// Prerun Pump
      A     DB145.DBX  172.6;
      AN    #S2I.SFM37.I00;
      A     #RRel;
      CLR   ;
      =     DB145.DBX  173.3;

// Return Pump
      AN    #Empty;
      A     #RRel;
      =     DB145.DBX  173.4;
      =     DB145.DBX   29.3;

// ---------------------------------------------------------------------------
// control modules (Own CM's)
      A     #ComCIP1;
      A     M    102.3;
      =     DB240.DBX  428.0;

      A     #ComCIP2;
      A     M    102.3;
      =     DB240.DBX  508.0;

      A     #ComCIP3;
      A     M    102.3;
      =     DB240.DBX  588.0;

// Trap Filter
      A     #S2I.SFM14.I01; // Yes
      A     M    102.3;
      CLR   ;
      =     DB240.DBX  188.0;
      =     DB240.DBX  348.0;

      A     #S2I.SFM14.I01; // Yes
      A     M    102.3;
      =     DB240.DBX  268.0;

// ---------------------------------------------------------------------------
// transition condition
//      A     #SubStepMaxD
//      =     "SOPD"


// subphase evaluation
      L     MW   110;
      JL    D500;
      JU    COMM; // subphase  0:
// ---------------------------------------------------------------------------
D500: SET   ;
      S     M    110.7; // Error unknown subphase
      JU    COMM;
NETWORK
TITLE =phase 36: CIP Drain
//SFM   Use                                 Datatype        UoM
//----+-------------------------------------------------------------------------
// 00 : Watch Dog Time                      Duration        Min
// 04 : Delay Empty                         Duration        #sec
X36:  SET   ;
// ---------------------------------------------------------------------------
// General CM evaluation
      CALL FC   140 (
           ChkType                  := 3,
           ChkOK                    := #ChkOK);

      AN    #ChkOK;
      S     M    120.3;

// ---------------------------------------------------------------------------
// general functions
      AN    M    121.2;
      A     M    102.3;
      =     #RRel;

// ---------------------------------------------------------------------------
// messages
// ---------------------------------------------------------------------------
// timer & counter
      A     DB145.DBX  458.5;
      A     M    102.0;
      =     M    130.3;


// ---------------------------------------------------------------------------
// pause timer
      ON    M    102.3;
      O     M    150.3;
      S     M    140.3; // Delay Empty

// ---------------------------------------------------------------------------
// communication

// ---------------------------------------------------------------------------
// control modules
      A     M    102.3;

// ---------------------------------------------------------------------------
// transition condition
      A     M    150.3;
      =     M    102.1;

// subphase evaluation
      L     MW   110;
      JL    D600;
      JU    COMM; // subphase  0:
// ---------------------------------------------------------------------------
D600: SET   ;
      S     M    110.7; // Error unknown subphase
      JU    COMM;
NETWORK
TITLE =phase 38: CIP Randvollstellung
//SFM   Use                                 Datatype        UoM
//----+-------------------------------------------------------------------------
// 00 : Watch Dog Time                      Duration        min
// 01 : Step Time                           Duration        min
// 04 : Delay Level                         Duration        s
// 15 : Amount                              Value           m3
// 17 : Level                               Value           l
// 22 : Agitator Speed                      Value           %
// 27 : CIP Prerun                          Enumeration     min
// 28 : CIP Return                          Enumeration     min
// 29 : CIP Pump Speed                      Value           %
// 34 : CIP Prerun Flow                     Value           m3/h
// 35 : CIP Prerun Pressure                 Value           bar
// 37 : CIP Pump Mode                       Enumeration     min
X38:  SET   ;
// ---------------------------------------------------------------------------
// General CM evaluation
      CALL FC   140 (
           ChkType                  := 3,
           ChkOK                    := #ChkOK);

      AN    #ChkOK;
      S     M    120.3;

// ---------------------------------------------------------------------------
// index evaluation: CIP Prerun
      CALL FC    45 (
           SFM                      := #U.Seq.SFM[27].Sp,
           Indexes                  := #S2I.SFM27);

// ---------------------------------------------------------------------------
// index evaluation: CIP Return
      CALL FC    45 (
           SFM                      := #U.Seq.SFM[28].Sp,
           Indexes                  := #S2I.SFM28);

// ---------------------------------------------------------------------------
// index evaluation: CIP Pump Mode
      CALL FC    45 (
           SFM                      := #U.Seq.SFM[37].Sp,
           Indexes                  := #S2I.SFM37);

// ---------------------------------------------------------------------------
// general functions
      AN    M    121.2;
      A     M    102.3;
      =     #RRel;

// Get Pushout Amount

      A     M    102.2;
      JCN   N381;
      L     #U.Seq.Prop.Val10;
      L     #U.Seq.SFM[15].Sp;
      +R    ;
      T     #U.Seq.SFM[15].Sp;
N381: NOP   0;

// CIP Unit
      AN    #ComCIP;
      ON    DB145.DBX  123.4;
      ON    DB145.DBX  123.5;
      JCN   x381;
      R     #RRel;
      L     949; // CIP Not Ready!
      T     MD    90;
x381: NOP   0;

// CIP Distribution Unit
      AN    #ComCIPDist;
      ON    DB145.DBX  411.4;
      ON    DB145.DBX  411.5;
      JCN   x382;
      R     #RRel;
      L     949; // CIP Partner Not Ready!
      T     MD    90;
x382: NOP   0;

// Partner Unit
      AN    #ComDST;
      ON    DB145.DBX  459.4;
      ON    DB145.DBX  459.5;
      JCN   x383;
      R     #RRel;
      L     903; // Partner Unit Not Ready!
      T     MD    90;
x383: NOP   0;

// CIP Signals ---
      CALL FC   716 (
           StepOnSFMSP              := #U.Seq.SFM[26].Sp,
           EmptySig                 := DB145.DBX  458.5,
           EmptyLevel               := TRUE,
           CIPPumpRun               := DB145.DBX  124.3,
           CIPReady                 := DB145.DBX  123.5,
           Empty                    := #Empty,
           TransCondOK              := M    102.1,
           RRel                     := #RRel);

      A     DB145.DBX  124.3;
      A     M    102.3;
      =     DB145.DBX   29.2;

// ---------------------------------------------------------------------------
// messages
// ---------------------------------------------------------------------------
// timer & counter
// Done in "CIPUnitC"
      A     M    102.3;
      =     M    130.0;
      =     M    131.6;

      A     DB145.DBX  458.2;
      A     M    102.3;
      =     M    130.3;

// ---------------------------------------------------------------------------
// communication
// Active, Prerun & Return
      A     M    102.0;
      =     DB145.DBX  171.4;
      =     DB145.DBX  172.6;
      R     DB145.DBX  172.7;

// Run Release
      A     #RRel;
      =     DB145.DBX  171.5;

// Prerun Pump
      A     DB145.DBX  172.6;
      AN    #S2I.SFM37.I00;
      A     #RRel;
      =     DB145.DBX  173.3;

// Return Pump
      AN    #Empty;
      A     #RRel;
      CLR   ;
      =     DB145.DBX  173.4;
      =     DB145.DBX   29.3;

// ---------------------------------------------------------------------------
// control modules (Own CM's)
      A     #ComCIP1;
      A     M    102.3;
      =     DB240.DBX  428.0;

      A     #ComCIP2;
      A     M    102.3;
      =     DB240.DBX  508.0;

      A     #ComCIP3;
      A     M    102.3;
      =     DB240.DBX  588.0;

// Trap Filter
      A     #S2I.SFM14.I01; // Yes
      A     M    102.3;
      CLR   ;
      =     DB240.DBX  188.0;
      =     DB240.DBX  348.0;

      A     #S2I.SFM14.I01; // Yes
      A     M    102.3;
      =     DB240.DBX  268.0;

// ---------------------------------------------------------------------------
// transition condition
      A     M    150.3;
      =     M    102.1;


// Nach Randvollstellung nach "CIP Ende"
      L     #U.Seq.StepMax; // CIP Ende = letzter Schritt
      T     MW   106;

// subphase evaluation
      L     MW   110;
      JL    D800;
      JU    COMM; // subphase  0:
// ---------------------------------------------------------------------------
D800: SET   ;
      S     M    110.7; // Error unknown subphase
      JU    COMM;
NETWORK
TITLE =phase 39: CIP Rinsing from RWT
//SFM   Use                                 Datatype        UoM
//----+-------------------------------------------------------------------------
// 00 : Watch Dog Time                      Duration        min
// 01 : Step Time                           Duration        min
// 05 : Substep Time                        Duration        s
// 06 : Delay Switchpoint                   Duration        s
// 15 : Amount                              Value           m3
// 27 : CIP Prerun                          Enumeration     min
// 28 : CIP Return                          Enumeration     min
// 29 : CIP Pump Speed                      Value           %
// 30 : CIP Return Temperature              Value           °C
// 32 : CIP Return Conductivity             Value           mS
// 34 : CIP Prerun Flow                     Value           m3/h
// 35 : CIP Prerun Pressure                 Value           bar
// 37 : CIP Pump Mode                       Enumeration     min
// 59 : Interval Counter                    Value           No.
X39:  SET   ;
// ---------------------------------------------------------------------------
// General CM evaluation
      CALL FC   140 (
           ChkType                  := 3,
           ChkOK                    := #ChkOK);

      AN    #ChkOK;
      S     M    120.3;

// ---------------------------------------------------------------------------
// index evaluation: CIP Prerun
      CALL FC    45 (
           SFM                      := #U.Seq.SFM[27].Sp,
           Indexes                  := #S2I.SFM27);

// ---------------------------------------------------------------------------
// index evaluation: CIP Return
      CALL FC    45 (
           SFM                      := #U.Seq.SFM[28].Sp,
           Indexes                  := #S2I.SFM28);

// ---------------------------------------------------------------------------
// index evaluation: CIP Pump Mode
      CALL FC    45 (
           SFM                      := #U.Seq.SFM[37].Sp,
           Indexes                  := #S2I.SFM37);

// ---------------------------------------------------------------------------
// general functions
      AN    M    121.2;
      A     M    102.3;
      =     #RRel;

// CIP Unit
      AN    #ComCIP;
      ON    DB145.DBX  123.4;
      ON    DB145.DBX  123.5;
      JCN   x391;
      R     #RRel;
      L     949; // CIP Not Ready!
      T     MD    90;
x391: NOP   0;

// CIP Distribution Unit
      AN    #ComCIPDist;
      ON    DB145.DBX  411.4;
      ON    DB145.DBX  411.5;
      JCN   x392;
      R     #RRel;
      L     949; // CIP Partner Not Ready!
      T     MD    90;
x392: NOP   0;

// Partner Unit
      AN    #ComDST;
      ON    DB145.DBX  459.4;
      ON    DB145.DBX  459.5;
      JCN   x393;
      R     #RRel;
      L     903; // Partner Unit Not Ready!
      T     MD    90;
x393: NOP   0;

// CIP Signals ---
      CALL FC   716 (
           StepOnSFMSP              := #U.Seq.SFM[26].Sp,
           EmptySig                 := DB145.DBX  458.5,
           EmptyLevel               := TRUE,
           CIPPumpRun               := DB145.DBX  124.3,
           CIPReady                 := DB145.DBX  123.5,
           Empty                    := #Empty,
           TransCondOK              := M    102.1,
           RRel                     := #RRel);


      A     DB145.DBX  124.3;
      A     M    102.3;
      =     DB145.DBX   29.2;



// ---------------------------------------------------------------------------
// messages
// ---------------------------------------------------------------------------
// timer & counter
// Done in "CIPUnitC"

// ---------------------------------------------------------------------------
// pause timer
      ON    M    102.3;
      O     M    150.0;
      S     M    140.0; // Step Time

      ON    M    102.3;
      O     M    150.5;
      S     M    140.5; // Delay Switchpoint

// ---------------------------------------------------------------------------
// communication
// Active, Prerun & Return
      A     M    102.0;
      =     DB145.DBX  171.4;
      =     DB145.DBX  172.7;
      =     DB145.DBX  172.6;

// Run Release
      A     #RRel;
      =     DB145.DBX  171.5;

// Prerun Pump
      A     DB145.DBX  459.5;
      A     DB145.DBX  172.6;
      AN    #S2I.SFM37.I00;
      A     #RRel;
      =     DB145.DBX  173.3;

// Return Pump
      AN    #Empty;
      A     #RRel;
      =     DB145.DBX  173.4;
      =     DB145.DBX   29.3;

// Mit Abluaf
      AN    M    157.2;
      A     M    102.0;
      =     DB145.DBX   29.5;

// ---------------------------------------------------------------------------
// control modules (Own CM's)
      A     #ComCIP1;
      A     M    102.3;
      =     DB240.DBX  428.0;

      A     #ComCIP2;
      A     M    102.3;
      =     DB240.DBX  508.0;

      A     #ComCIP3;
      A     M    102.3;
      =     DB240.DBX  588.0;

// Trap Filter
      A     #S2I.SFM14.I01; // Yes
      A     M    102.3;
      CLR   ;
      =     DB240.DBX  188.0;
      =     DB240.DBX  348.0;

      A     #S2I.SFM14.I01; // Yes
      A     M    102.3;
      =     DB240.DBX  268.0;

// ---------------------------------------------------------------------------
// transition condition
//      A     #SubStepMaxD
//      =     "SOPD"

// ---------------------------------------------------------------------------
// ---------------------------------------------------------------------------
// subphase repeat function
      A     #SubStepMax;
      JCN   Y39;
      L     1;
      T     MW   116;
Y39:  SET   ;

      A     #SubStepMax;
      AN    M    103.0;
      JCN   Y39a;
      L     #U.Seq.SFM[59].Val; // Increment Interval Counter
      L     1.000000e+000;
      +R    ;
      T     #U.Seq.SFM[59].Val;
Y39a: SET   ;
      A     M    102.2;
      ON    M    102.0;
      JCN   In2R; // Reset Interval Counter at Start and End Of Phase
      L     0.000000e+000;
      T     #U.Seq.SFM[59].Val;
In2R: NOP   0;

// subphase evaluation
      L     MW   110;
      JL    D900;
      JU    COMM; // subphase  0:
      JU    D901; // subphase  1: Pause
      JU    D902; // subphase  2: Main
      JU    D903; // subphase  3: Expulse
      JU    D904; // subphase  4: Seat Lift
      JU    D900; // subphase  5:
      JU    D906; // subphase  6: Shaft Rinse
      JU    D907; // subphase  7: Drain
// ---------------------------------------------------------------------------
D900: SET   ;
      S     M    110.7; // Error unknown subphase
      JU    COMM;

// subphase 1: Pause
D901: SET   ;

      A     M    103.0;
      R     DB145.DBX  173.3;

// -------------------------------------------------
// subphase timer & counter
      A     M    103.0;
      =     M    130.4; // Substep Time
// -------------------------------------------------
// subphase actuator

// -------------------------------------------------
// subphase transition
      A     M    150.3; // Delay Level
      A     M    130.3;
      O     M    150.4; // Substep Time Done
      =     M    103.1;
      JU    COMM;

// subphase 2: Main
D902: SET   ;

// -------------------------------------------------
// subphase timer & counter
      A     M    103.0;
      =     M    130.4; // Substep Time

// -------------------------------------------------
// subphase actuator
      A     M    103.3;


// -------------------------------------------------
// subphase transition
      A     M    150.4; // Substep Time Done
      =     M    103.1;
      JU    COMM;

// subphase 3: Expulse
D903: SET   ;

// -------------------------------------------------
// subphase timer & counter
      A     M    103.0;

// -------------------------------------------------
// subphase actuator
      A     M    103.3;

// -------------------------------------------------
// subphase transition
      CLR   ;
      =     M    103.1;
      JU    COMM;

// subphase 4: Seat Lift
D904: SET   ;

// -------------------------------------------------
// subphase timer & counter
      A     M    103.0;

// -------------------------------------------------
// subphase actuator
      A     M    103.3;

// -------------------------------------------------
// subphase transition
      SET   ;
      =     M    103.1;
      JU    COMM;

// subphase 6: Shaft Rinse
D906: SET   ;

// -------------------------------------------------
// subphase timer & counter
      A     M    103.0;
      =     M    130.4; // Substep Time

// -------------------------------------------------
// subphase actuator
      A     M    103.3;
      =     DB240.DBX  668.0;

// -------------------------------------------------
// subphase transition
      A     M    150.4; // Substep Time Done
      O     M    157.2; // Interval Counter Done
      =     M    103.1;
      JU    COMM;

// subphase 7: Drain
D907: SET   ;

// -------------------------------------------------
// subphase timer & counter
      A     M    103.0;
      =     M    130.4; // Substep Time

// -------------------------------------------------
// subphase actuator
      A     M    103.3;
      R     DB145.DBX  173.6; // Req Drain RV1_RS
      R     DB145.DBX   29.6; // Req Common Drain
      R     DB2990.DBX  268.0;

// -------------------------------------------------
// subphase transition
      A     M    150.4; // Substep Time Done
      O     M    157.2; // Interval Counter Done
      =     M    103.1;
      JU    COMM;
NETWORK
TITLE =phase 40: CIP End
//SFM   Use                                 Datatype        UoM
//----+-------------------------------------------------------------------------
// 00 : Watch Dog Time                      Duration        min
X40:  SET   ;
// ---------------------------------------------------------------------------
// General CM evaluation
      CALL FC   140 (
           ChkType                  := 3,
           ChkOK                    := #ChkOK);

      AN    #ChkOK;
      S     M    120.3;

// ---------------------------------------------------------------------------
// general functions
//      AN    "SOSTAl"
      A     M    102.3;
      =     #RRel;

// CIP Signals ---
      CALL FC   716 (
           StepOnSFMSP              := 0.000000e+000,
           EmptySig                 := FALSE,
           EmptyLevel               := FALSE,
           CIPPumpRun               := FALSE,
           CIPReady                 := FALSE,
           Empty                    := #xTmp,
           TransCondOK              := #xTmp,
           RRel                     := #RRel);

// ---------------------------------------------------------------------------
// communication
      A     M    102.0;
      =     DB145.DBX   29.7;
      =     DB145.DBX  173.7;

// ---------------------------------------------------------------------------
// transition condition
      AN    #ComCIP;
      AN    #ComCIPDist;
      AN    #ComDST;
      =     M    102.1;


// subphase evaluation
      L     MW   110;
      JL    E000;
      JU    COMM; // subphase  0:
// ---------------------------------------------------------------------------
E000: SET   ;
      S     M    110.7; // Error unknown subphase
      JU    COMM;

NETWORK
TITLE =End Of Sequence Organisation

COMM: SET   ;

// ---------------------------------------------------------------------------
// pause timer unit parameter


NETWORK
TITLE =General Post Phase Controls

      NOP   0;

// ---------------------------------------------------------------------------
// general postphase controls

      L     #U.Seq.PrId;
      L     DB1945.DBD   10;
      ==D   ;
      A(    ;
      L     0;
      >D    ;
      )     ;
      JCN   CIP1;

      CALL SFC   20 (
           SRCBLK                   := DB145.ToCIP,
           RET_VAL                  := #iTmp,
           DSTBLK                   := DB502.ToCIP1);

CIP1: NOP   0;

      L     #U.Seq.PrId;
      L     DB1955.DBD   10;
      ==D   ;
      A(    ;
      L     0;
      >D    ;
      )     ;
      JCN   CIP2;

      CALL SFC   20 (
           SRCBLK                   := DB145.ToCIP,
           RET_VAL                  := #iTmp,
           DSTBLK                   := DB502.ToCIP2);
CIP2: NOP   0;

      L     #U.Seq.PrId;
      L     DB1965.DBD   10;
      ==D   ;
      A(    ;
      L     0;
      >D    ;
      )     ;
      JCN   CIP3;

      CALL SFC   20 (
           SRCBLK                   := DB145.ToCIP,
           RET_VAL                  := #iTmp,
           DSTBLK                   := DB502.ToCIP3);

CIP3: NOP   0;


// Check Selection / Material -----------------------------------------------
      L     0;
      L     DB145.DBD  222; // 1. Tank
      <R    ;
      JCN   MCk1;
      L     #U.Seq.SFM[42].Sp;
      <>R   ;
      S     M    120.3;
      JCN   MCk0;
      L     910;
      T     MD    80;
MCk0: NOP   0;
      L     0;
      L     DB145.DBD  270; // 1. Tank
      <R    ;
      JCN   MCk1;
      L     #U.Seq.SFM[42].Sp;
      <>R   ;
      JCN   MCk1;
      L     910;
      T     MD    90;
MCk1: NOP   0;
      L     0;
      L     DB145.DBD  318; // 2. Tank
      <R    ;
      JCN   MCk2;
      L     #U.Seq.SFM[42].Sp;
      <>R   ;
      JCN   MCk2;
      L     910;
      T     MD    90;
MCk2: NOP   0;
      L     0;
      L     DB145.DBD  366; // 3. Tank
      <R    ;
      JCN   MCk3;
      L     #U.Seq.SFM[42].Sp;
      <>R   ;
      JCN   MCk3;
      L     910;
      T     MD    90;
MCk3: NOP   0;

      L     #U.Seq.SFM[11].Sp;
      L     #U.Seq.SFM[12].Sp;
      OD    ;
      L     #U.Seq.SFM[13].Sp;
      OD    ;
      L     0;
      >R    ;
      O     M    120.7;
      O     #CIP;
      JC    TSel;
      L     906; // "Source not Selected"
      T     MD    90;
TSel: NOP   0;

NETWORK
TITLE =Process Status Management

      NOP   0;
// ---------------------------------------------------------------------------
// Signal Control

      OPN   DB   500;
      L     #UnitNo;
      L     32; //U Structure Length
      *I    ;
      L     20; //DB Heading Offset
      +I    ;
      SLD   3;
      LAR2  ;

// -------------------------------------------------
// Maintenance
      A     #U.Seq.Switch.Sw31;
      OPN   DB   500;
      =     DBX [AR2,P#0.0]; //"PStatD".U[#UnitNo].MTNC
// -------------------------------------------------
// CIP Required
// -------------------------------------------------
// CIP Active
// -------------------------------------------------
// CIP Clean
// -------------------------------------------------
// SIP Required
// -------------------------------------------------
// SIP Active
// -------------------------------------------------
// SIP Clean
// -------------------------------------------------
// Full
      A     DB145.DBX   26.2;
      OPN   DB   500;
      =     DBX [AR2,P#0.7]; //"PStatD".U[#UnitNo].FULL
// -------------------------------------------------
// Filling
      A     DB145.DBX   26.1;
      OPN   DB   500;
      =     DBX [AR2,P#1.0]; //"PStatD".U[#UnitNo].FILL
// -------------------------------------------------
// Ready For Filling
      A     DB145.DBX   26.0;
      OPN   DB   500;
      =     DBX [AR2,P#1.1]; //"PStatD".U[#UnitNo].RFFI
// -------------------------------------------------
// Empty
      A     DB145.DBX   26.5;
      OPN   DB   500;
      =     DBX [AR2,P#1.2]; //"PStatD".U[#UnitNo].EMTY
// -------------------------------------------------
// Emptying
      A     DB145.DBX   26.4;
      OPN   DB   500;
      =     DBX [AR2,P#1.3]; //"PStatD".U[#UnitNo].EMTI
// -------------------------------------------------
// Ready For Emptying
      A     DB145.DBX   26.3;
      OPN   DB   500;
      =     DBX [AR2,P#1.4]; //"PStatD".U[#UnitNo].RFEM
// -------------------------------------------------
// Reserved
//      A     #ComXYZ
//      OPN   "PStatD"
//      =     DBX [AR2,P#1.5]             //"PStatD".U[#UnitNo].RESV
// -------------------------------------------------
// Production
// -------------------------------------------------
// Used

// -------------------------------------------------
// PStat Function Call

      CALL FC   500 (
           UnitNo                   := #UnitNo,
           PStatModVal              := DB245.DBD  234);



NETWORK
TITLE =Unit Hold Request and Messages

      SET   ;

// ---------------------------------------------------------------------------
// Set unit to "hold" if maintenance
      AN    #U.Seq.Switch.Sw31; // maintenance !
      JC    NCO1;
      S     M    120.3;
      L     998; // "Unit in maintenance !"
      T     MD    90;

// ---------------------------------------------------------------------------
// Set unit to "hold" if emergency stop
NCO1: A     #EStopOK;
      JC    NCO2;
      S     M    120.3;
      L     999; // "Emergency stop !"
      T     MD    90;
NCO2: NOP   0;

// ---------------------------------------------------------------------------
// Check Partner
      AN    #S2I.SFM10.I00;
      AN    #U.Seq.PO.B22;
      AN    #U.Seq.Step0;
      AN    #CIP;
      =     #xTmp;


      AN    DB145.DBX  218.3;
      AN    DB145.DBX  218.4;
      A     #xTmp;
      JCN   NC03;
      L     904; // "Source Not Ready!
      T     MD    90;
NC03: NOP   0;

      AN    DB145.DBX  218.3;
      ON    DB145.DBX  218.4;
      AN    #ComSRC;
      AN    #U.Seq.Step0;
      AN    #U.Seq.PO.B22;
      AN    #CIP;
      JCN   NC06;
      L     909; // Source for Material not found
      T     MD    90;
NC06: NOP   0;

      AN    #S2I.SFM14.I02;
      AN    #U.Seq.Step0;
      AN    #CIP;
      CLR   ;
      JCN   NC04;
      L     903; // Partner not Ready
      T     MD    90;
NC04: NOP   0;

      AN    DB145.DBX  458.0; // Water Tank Ready
      AN    DB145.DBX  458.1;
      AN    #U.Seq.Step0;
      AN    #U.Seq.PO.B3;
      AN    #CIP;
      CLR   ;
      JCN   NC05;
      L     903; // Destination not Ready
      T     MD    90;
NC05: NOP   0;






END_FUNCTION_BLOCK

FUNCTION_BLOCK FB 143
TITLE =C04: Water Transfer Plant x
AUTHOR : Woermann
FAMILY : BOTEC_F1
NAME : C04E
VERSION : 1.2
CODE_VERSION1


VAR
  U : UDT 141;
END_VAR
VAR_TEMP
  CIP : BOOL ;	//CIP active
  UNIM : BOOL ;	//Unit Not In Maintenance
  GenRel : BOOL ;	//general OK (emergency and maintenance OK)
  EStopOK : BOOL ;	//emergency OK
  UnitNo : INT ;	//unit number
  xTmp : BOOL ;	//Temporary Bool
  iTmp : INT ;	//Temporary INT
  rTmp : REAL ;	//Temporary REAL
  dTmp : DINT ;	//Temporary DINT (free for general use)
  RetValInt : INT ;	//return value
  ComCIP1 : BOOL ;	//CIP1 in use
  ComCIP3 : BOOL ;	//CIP3 in use
END_VAR
BEGIN
NETWORK
TITLE =General

      SET   ;
// Simulation ---------------------------------------------------------------
      A     #U.Seq.User.Bit63;
      CC    FB   149; // "C04Sim"
      A     #U.Seq.Sim;
      =     #U.Seq.User.Bit63; //Help bit for simulation

// get unit number ----------------------------------------------------------
      L     #U.Seq.UnitNo;
      T     #UnitNo;

// CIP ----------------------------------------------------------------------
      L     #U.Seq.ProgNo;
      L     0;
      <D    ;
      =     #CIP;

// emergency OK -------------------------------------------------------------
      A     DB145.DBX   27.0; //Emergency Stop OK
      =     #EStopOK;

// Write Unit in Maintenance ------------------------------------------------

      AN    #U.Seq.Switch.Sw31;
      =     #UNIM;

// emergency and maintenance OK ---------------------------------------------
      A     #EStopOK;
      A     #UNIM;
      =     #GenRel;

// communication ------------------------------------------------------------
      UC    FB   145; // C04Com

NETWORK
TITLE =Universal Value

      NOP   0;

// ----------------------------------------------------------
// unv001 Process Status
// ----------------------------------------------------------
// process value to UnV
//      L     0.000000e+000
//      T     "C04UnVD".unv001.ValExt

// ----------------------------------------------------------
// unv002 Universal Value 02
// ----------------------------------------------------------
// process value to UnV
//      L     0.000000e+000
//      T     "C04UnVD".unv002.ValExt

// ----------------------------------------------------------
// unv003 Universal Value 03
// ----------------------------------------------------------
// process value to UnV
//      L     0.000000e+000
//      T     "C04UnVD".unv003.ValExt

// ----------------------------------------------------------
// unv004 Universal Value 04
// ----------------------------------------------------------
// process value to UnV
//      L     0.000000e+000
//      T     "C04UnVD".unv004.ValExt

NETWORK
TITLE =Special Input

      NOP   0;

// ----------------------------------------------------------
// RM_KEG_V14 KEG_V14
// ----------------------------------------------------------
      CLR   ;
      =     DB241.DBX   81.4;
      =     DB241.DBX   81.5;

NETWORK
TITLE =Messages

      NOP   0;

// ----------------------------------------------------------
// msg001 Message 01
// ----------------------------------------------------------
      SET   ;
      R     DB247.DBX   80.7;
      =     DB247.DBX   81.4;

      CLR   ;
      =     DB247.DBX   82.7;

// ----------------------------------------------------------
// msg002 Message 02
// ----------------------------------------------------------
      SET   ;
      R     DB247.DBX  140.7;
      =     DB247.DBX  141.4;

      CLR   ;
      =     DB247.DBX  142.7;

// ----------------------------------------------------------
// msg003 Message 03
// ----------------------------------------------------------
      SET   ;
      R     DB247.DBX  200.7;
      =     DB247.DBX  201.4;

      CLR   ;
      =     DB247.DBX  202.7;

NETWORK
TITLE =Sequence organisation


// SFM supply ----------------------------------------------------------------


NETWORK
TITLE =Auto / Manual

      SET   ;
      AN    M    122.2;
      JC    MODE;
      AN    M    120.1;

// assign actuator mode
      AN    M    120.1;
      =     DB240.DBX  105.4;
      =     DB240.DBX  185.4;
      =     DB240.DBX  265.4;
      =     DB240.DBX  345.4;
      =     DB240.DBX  425.4;
      =     DB240.DBX  505.4;
      =     DB240.DBX  585.4;
      =     DB240.DBX  665.4;
      =     DB240.DBX  745.4;
      =     DB240.DBX  825.4;
MODE: SET   ;

NETWORK
TITLE =Wasserpumpe
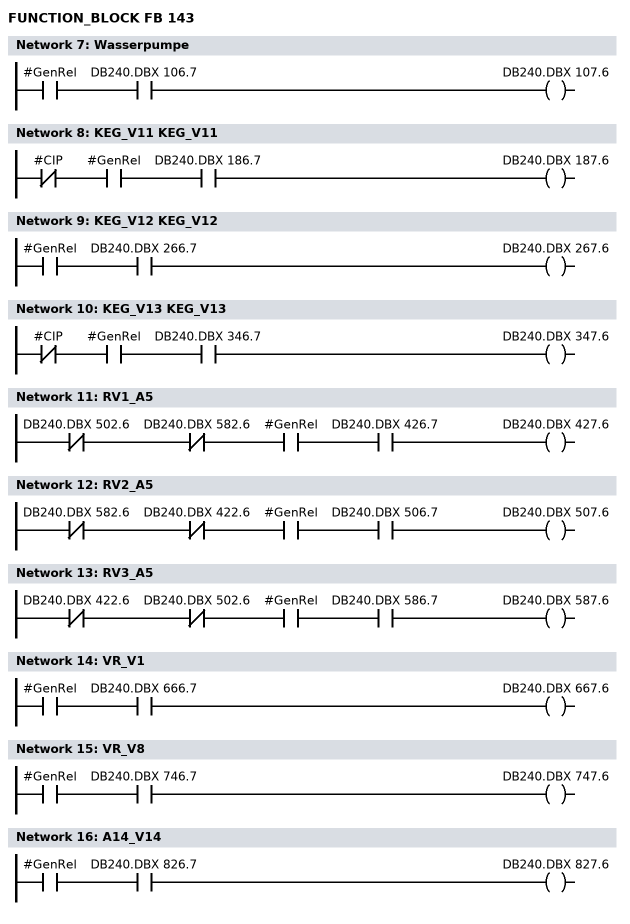

      A     #GenRel;
      A     DB240.DBX  106.7;
      =     DB240.DBX  107.6;

NETWORK
TITLE =KEG_V11 KEG_V11

      AN    #CIP;
      A     #GenRel;
      A     DB240.DBX  186.7;
      =     DB240.DBX  187.6;
NETWORK
TITLE =KEG_V12 KEG_V12

      A     #GenRel;
      A     DB240.DBX  266.7;
      =     DB240.DBX  267.6;
NETWORK
TITLE =KEG_V13 KEG_V13

      AN    #CIP;
      A     #GenRel;
      A     DB240.DBX  346.7;
      =     DB240.DBX  347.6;
NETWORK
TITLE =RV1_A5

      AN    DB240.DBX  502.6;
      AN    DB240.DBX  582.6;

      A     #GenRel;
      A     DB240.DBX  426.7;
      =     DB240.DBX  427.6;

NETWORK
TITLE =RV2_A5

      AN    DB240.DBX  582.6;
      AN    DB240.DBX  422.6;

      A     #GenRel;
      A     DB240.DBX  506.7;
      =     DB240.DBX  507.6;

NETWORK
TITLE =RV3_A5

      AN    DB240.DBX  422.6;
      AN    DB240.DBX  502.6;

      A     #GenRel;
      A     DB240.DBX  586.7;
      =     DB240.DBX  587.6;

NETWORK
TITLE =VR_V1

      A     #GenRel;
      A     DB240.DBX  666.7;
      =     DB240.DBX  667.6;

NETWORK
TITLE =VR_V8

      A     #GenRel;
      A     DB240.DBX  746.7;
      =     DB240.DBX  747.6;

NETWORK
TITLE =A14_V14

      A     #GenRel;
      A     DB240.DBX  826.7;
      =     DB240.DBX  827.6;

END_FUNCTION_BLOCK

FUNCTION_BLOCK FB 145
TITLE =C04: Water Transfer Plant x
AUTHOR : Woermann
FAMILY : BOTEC_F1
NAME : C04Comm
VERSION : 0.1
CODE_VERSION1


VAR
  U : UDT 141;
END_VAR
VAR_TEMP
  iRetVal : INT ;	//return value as integer
  wRetVal : WORD ;	//return value as word
  Run : BOOL ;	//Unit in "RUN" mode
  EStopOK : BOOL ;	//Emergency Stop OK
  CIP : BOOL ;	//CIP Program Selected
  ComCIP : BOOL ;	//Communication with CIP Active
  xTmp : BOOL ;	//Temporary BOOL (free for general use)
  iTmp : INT ;	//Temporary INT (free for general use)
  rTmp : REAL ;	//Temporary REAL (free for general use)
  dTmp : DINT ;	//Temporary DINT (free for general use)
  UnitNo : INT ;	//Unit Number
  EquipmentID : INT ;	//Equipment ID
  Prid : DINT ;	//Process ID
  SFM36 : STRUCT 	//CIP Pump Mode
   I00 : BOOL ;	// Off
   I01 : BOOL ;	// Flow
   I02 : BOOL ;	// Pressure
   I03 : BOOL ;	// Fix Speed
   I04 : BOOL ;
   I05 : BOOL ;
   I06 : BOOL ;
   I07 : BOOL ;
   I08 : BOOL ;
   I09 : BOOL ;
   I10 : BOOL ;
   I11 : BOOL ;
   I12 : BOOL ;
   I13 : BOOL ;
   I14 : BOOL ;
   I15 : BOOL ;
   I16 : BOOL ;
   I17 : BOOL ;
   I18 : BOOL ;
   I19 : BOOL ;
   I20 : BOOL ;
   I21 : BOOL ;
   I22 : BOOL ;
   I23 : BOOL ;
   I24 : BOOL ;
   I25 : BOOL ;
   I26 : BOOL ;
   I27 : BOOL ;
   I28 : BOOL ;
   I29 : BOOL ;
   I30 : BOOL ;
   I31 : BOOL ;
  END_STRUCT ;
  iPLC : INT ;
  iUnit : INT ;
  rUnitNo : REAL ;
  DSTUnit : INT ;	//Destination Unit
  SRCUnit : INT ;
  STBYUnit : INT ;
  rEquipmentID : REAL ;
  dst0 : BOOL ;	//No Destination Selected
END_VAR
BEGIN
NETWORK
TITLE =general

      SET   ;

// unit & equipment number ---------------------------------------------------
      L     #U.Seq.UnitNo;
      T     #UnitNo;

      L     DB145.DBW   14;
      L     1000;
      *I    ;
      L     #UnitNo;
      +I    ;
      T     #EquipmentID;

      L     #EquipmentID;
      ITD   ;
      DTR   ;
      T     #rEquipmentID;

// CIP ----------------------------------------------------------------------
      L     DB145.DBW   18;
      L     0;
      <I    ;
      =     #CIP;

// Communicating Units-------------------------------------------------------
      L     DB145.DBD   10;
      L     DB145.DBD  106;
      ==D   ;
      =     #ComCIP;


NETWORK
TITLE =read other unit's data

      SET   ;

// ... General Unit ----------/

      CALL SFC   20 (
           SRCBLK                   := DB1995.Own,
           RET_VAL                  := #iRetVal,
           DSTBLK                   := DB145.GEN);

// emergency OK -------------------------------------------------------------
      A     DB145.DBX   75.0; //General Emergency Stop OK
      =     #EStopOK;


//----------------------------------------
// Communication Water Tank
//----------------------------------------

// Current Tank ----------------------------

      L     #U.Seq.SFM[10].Sp;
      L     0.000000e+000;
      >R    ;
      JCN   N201;

      CALL FC   950 (
           EquipmentNo              := #U.Seq.SFM[10].Sp,
           PLCNo                    := #iPLC,
           UnitNo                   := #iUnit);

      CALL FC   563 (
           ActReq                   := M    101.0,
           PLCNo                    := #iPLC,
           SourceUnitNo             := #iUnit,
           IsTUnit                  := FALSE,
           DstComDRec               := DB145.SRC,
           RET_VAL                  := #wRetVal);
      JU    N2x1;
N201: NOP   0;
      L     0;
      T     #rTmp;
      CALL SFC   21 (
           BVAL                     := #rTmp,
           RET_VAL                  := #iTmp,
           BLK                      := DB145.SRC);
N2x1: NOP   0;

// Priority 1 -----------------------------

      L     #U.Seq.SFM[11].Sp;
      L     0.000000e+000;
      >R    ;
      JCN   N202;


      CALL FC   950 (
           EquipmentNo              := #U.Seq.SFM[11].Sp,
           PLCNo                    := #iPLC,
           UnitNo                   := #iUnit);

      CALL FC   563 (
           ActReq                   := M    101.0,
           PLCNo                    := #iPLC,
           SourceUnitNo             := #iUnit,
           IsTUnit                  := FALSE,
           DstComDRec               := DB145.SRC1,
           RET_VAL                  := #wRetVal);
      JU    N2x2;
N202: NOP   0;
      L     0;
      T     #rTmp;
      CALL SFC   21 (
           BVAL                     := #rTmp,
           RET_VAL                  := #iTmp,
           BLK                      := DB145.SRC1);
N2x2: NOP   0;

// Priority 2 ----------------------------

      L     #U.Seq.SFM[12].Sp;
      L     0.000000e+000;
      >R    ;
      JCN   N203;


      CALL FC   950 (
           EquipmentNo              := #U.Seq.SFM[12].Sp,
           PLCNo                    := #iPLC,
           UnitNo                   := #iUnit);

      CALL FC   563 (
           ActReq                   := M    101.0,
           PLCNo                    := #iPLC,
           SourceUnitNo             := #iUnit,
           IsTUnit                  := FALSE,
           DstComDRec               := DB145.SRC2,
           RET_VAL                  := #wRetVal);
      JU    N2x3;
N203: NOP   0;
      L     0;
      T     #rTmp;
      CALL SFC   21 (
           BVAL                     := #rTmp,
           RET_VAL                  := #iTmp,
           BLK                      := DB145.SRC2);
N2x3: NOP   0;

// Priority 3 ----------------------------

      L     #U.Seq.SFM[13].Sp;
      L     0.000000e+000;
      >R    ;
      JCN   N204;


      CALL FC   950 (
           EquipmentNo              := #U.Seq.SFM[13].Sp,
           PLCNo                    := #iPLC,
           UnitNo                   := #iUnit);

      CALL FC   563 (
           ActReq                   := M    101.0,
           PLCNo                    := #iPLC,
           SourceUnitNo             := #iUnit,
           IsTUnit                  := FALSE,
           DstComDRec               := DB145.SRC3,
           RET_VAL                  := #wRetVal);
      JU    N2x4;
N204: NOP   0;
      L     0;
      T     #rTmp;
      CALL SFC   21 (
           BVAL                     := #rTmp,
           RET_VAL                  := #iTmp,
           BLK                      := DB145.SRC3);
N2x4: NOP   0;

//----------------------------------------
// Communication Packaging Plant
//----------------------------------------
      L     #U.Seq.Prop.Index0; // Destination
      ITD   ;
      DTR   ;
      T     #rTmp;

      CALL FC   950 (
           EquipmentNo              := #rTmp,
           PLCNo                    := #iPLC,
           UnitNo                   := #iUnit);


      CALL FC   563 (
           ActReq                   := M    101.0,
           PLCNo                    := #iPLC,
           SourceUnitNo             := #iUnit,
           IsTUnit                  := FALSE,
           DstComDRec               := DB145.DST,
           RET_VAL                  := #wRetVal);

NETWORK
TITLE =external releases

      SET   ;
      =     DB240.DBX  106.7;
      =     DB240.DBX  186.7;
      =     DB240.DBX  266.7;
      =     DB240.DBX  346.7;
      =     DB240.DBX  426.7;
      =     DB240.DBX  506.7;
      =     DB240.DBX  586.7;
      =     DB240.DBX  666.7;
      =     DB240.DBX  746.7;
      =     DB240.DBX  826.7;

NETWORK
TITLE =write own unit data

      SET   ;

//-- CIP Communication ---------------------------------------
      AN    #U.Seq.Step0;
      AN    #U.Seq.PO.B30; // CIP Active (Slave)
      O(    ;
      A     #U.Seq.PO.B3; // Prerinse
      L     DB145.DBD   10;
      L     DB145.DBD  394;
      ==I   ;
      )     ;
//    A     #ComCIP
      JCN   NCIP;
//Conductivity CIP Return
      L     DB145.DBD  150;
      T     #U.Seq.SFM[32].Val;

//Temperature CIP Return
      L     DB145.DBD  146;
      T     #U.Seq.SFM[30].Val;

//CIP Prerun Pump SP

      CALL FC    45 (
           SFM                      := #U.Seq.SFM[36].Sp,
           Indexes                  := #SFM36);


      L     0.000000e+000;
      A     #SFM36.I01;
      =     DB145.DBX  171.7;
      JCN   pfc;
      L     #U.Seq.SFM[34].Sp;
pfc:  NOP   0;
      A     #SFM36.I02;
      =     DB145.DBX  172.0;
      JCN   ppc;
      L     #U.Seq.SFM[35].Sp;
ppc:  NOP   0;
      A     #SFM36.I03;
      =     DB145.DBX  171.6;
      JCN   pxc;
      L     #U.Seq.SFM[29].Sp;
pxc:  NOP   0;
      T     DB145.DBD  182;

// CIP Prerun Temperature
      L     #U.Seq.SFM[36].Sp;
      T     DB145.DBD  182;

//CIP Return
      L     #U.Seq.SFM[28].Sp;
      T     DB145.DBD  186;
      L     DB145.DBD  138;
      T     #U.Seq.SFM[28].Val;

//CIP Prerun
      L     #U.Seq.SFM[27].Sp;
      T     DB145.DBD  190;
      L     DB145.DBD  142;
      T     #U.Seq.SFM[27].Val;

// Write Own Data to CIP
      L     DB145.DBD   10;
      T     DB145.DBD  154;

      L     DB145.DBW   14;
      T     DB145.DBW  158;

      L     DB145.DBW   16;
      T     DB145.DBW  160;

      L     DB145.DBW   18;
      T     DB145.DBW  162;

      L     DB145.DBW   20;
      T     DB145.DBW  164;

      L     DB145.DBW   22;
      T     DB145.DBW  166;

      A     DB145.DBX   24.0;
      =     DB145.DBX  168.0;

      A     DB145.DBX   24.1;
      =     DB145.DBX  168.1;

      A     DB145.DBX   24.2;
      =     DB145.DBX  168.2;

      A     DB145.DBX   24.3;
      =     DB145.DBX  168.3;

      A     DB145.DBX   24.4;
      =     DB145.DBX  168.4;

      A     DB145.DBX   24.5;
      =     DB145.DBX  168.5;

      A     DB145.DBX   24.6;
      =     DB145.DBX  168.6;

      A     DB145.DBX   24.7;
      =     DB145.DBX  168.7;

// Copy Data to CIP
//      CALL  "BLKMOV"
//       SRCBLK :="C04ComD".ToCIP
//       RET_VAL:=#iRetVal
//       DSTBLK :="C04ComD".ToCIP

NCIP: NOP   0;

//Empty Signal
//A     "C04SpID".SpI.Sig //!!!! Insert correct Empty Signal !!!
      CLR   ;
      =     DB145.DBX   26.5;

//Full Signal
//A     "C04SpID".SpI.Sig //!!!! Insert correct Full Signal !!!
      CLR   ;
      =     DB145.DBX   26.2;

//CIP Program Selected
      A     #CIP;
      =     DB145.DBX   27.1;

// Emergency Stop
      A     #EStopOK; //If needed add or replace with own SpI
      =     DB145.DBX   27.0; //Emergency Stop OK

      L     #U.Seq.SFM[42].Sp; // Material
      T     DB145.DBD   30;

      L     #U.Seq.SFM[10].Sp; // Current Water Tank Selection
      T     DB145.DBD   34;

      L     #U.Seq.SFM[11].Sp; // Priority 1
      T     DB145.DBD   38;

      L     #U.Seq.SFM[12].Sp; // Priority 2
      T     DB145.DBD   42;

      L     #U.Seq.SFM[13].Sp; // Priority 3
      T     DB145.DBD   46;

      L     DB145.DBD  138; // CIP Amount
      T     DB145.DBD   54; // CIP Amount


NETWORK
TITLE = read from other unit data

      L     0;
      T     #rTmp;



// ... CIP / CIP Distribution ------------- /
      L     #U.Seq.PrId;
      L     DB1945.DBD   10;
      ==D   ;
      A(    ;
      L     0;
      >D    ;
      )     ;
      JCN   CIP1;
      CALL FC   563 (
           ActReq                   := M    101.0,
           PLCNo                    := 3,
           SourceUnitNo             := 91,
           IsTUnit                  := FALSE,
           DstComDRec               := DB145.CIP,
           RET_VAL                  := #wRetVal);

      CALL FC   563 (
           ActReq                   := M    101.0,
           PLCNo                    := 3,
           SourceUnitNo             := 94,
           IsTUnit                  := FALSE,
           DstComDRec               := DB145.CIPDist,
           RET_VAL                  := #wRetVal);
      JU    NZ;
CIP1: NOP   0;


      L     #U.Seq.PrId;
      L     DB1955.DBD   10;
      ==D   ;
      A(    ;
      L     0;
      >D    ;
      )     ;
      JCN   CIP2;
      CALL FC   563 (
           ActReq                   := M    101.0,
           PLCNo                    := 3,
           SourceUnitNo             := 92,
           IsTUnit                  := FALSE,
           DstComDRec               := DB145.CIP,
           RET_VAL                  := #wRetVal);

      CALL FC   563 (
           ActReq                   := M    101.0,
           PLCNo                    := 3,
           SourceUnitNo             := 95,
           IsTUnit                  := FALSE,
           DstComDRec               := DB145.CIPDist,
           RET_VAL                  := #wRetVal);
      JU    NZ;
CIP2: NOP   0;

      L     #U.Seq.PrId;
      L     DB1965.DBD   10;
      ==D   ;
      A(    ;
      L     0;
      >D    ;
      )     ;
      JCN   CIP3;
      CALL FC   563 (
           ActReq                   := M    101.0,
           PLCNo                    := 3,
           SourceUnitNo             := 93,
           IsTUnit                  := FALSE,
           DstComDRec               := DB145.CIP,
           RET_VAL                  := #wRetVal);

      CALL FC   563 (
           ActReq                   := M    101.0,
           PLCNo                    := 3,
           SourceUnitNo             := 96,
           IsTUnit                  := FALSE,
           DstComDRec               := DB145.CIPDist,
           RET_VAL                  := #wRetVal);
      JU    NZ;
CIP3: NOP   0;



// Zero the data
      CALL SFC   21 (
           BVAL                     := #rTmp,
           RET_VAL                  := #iTmp,
           BLK                      := DB145.CIP);

      CALL SFC   21 (
           BVAL                     := #rTmp,
           RET_VAL                  := #iTmp,
           BLK                      := DB145.CIPDist);

NZ:   NOP   0;
END_FUNCTION_BLOCK

FUNCTION_BLOCK FB 149
TITLE =C04: Water Transfer Plant x
AUTHOR : Woermann
FAMILY : BOTEC_F1
NAME : C04Sim
VERSION : 0.1
CODE_VERSION1


VAR
  U : UDT 141;
END_VAR
VAR_TEMP
  CIP : BOOL ;	//CIP active
  xTmp : BOOL ;	//Temporary BOOL (free for general use)
  iTmp : INT ;	//Temporary INT (free for general use)
  rTmp : REAL ;	//Temporary REAL (free for general use)
  UnitNo : INT ;	//Unit Number
END_VAR
BEGIN
NETWORK
TITLE =General

      SET   ;
// get unit number ----------------------------------------------------------
      L     #U.Seq.UnitNo;
      T     #UnitNo;

// CIP ----------------------------------------------------------------------
      L     #U.Seq.ProgNo;
      L     0;
      <D    ;
      =     #CIP;

NETWORK
TITLE =Actuator

      A     #U.Seq.Sim;
      =     DB240.DBX  105.3;
      =     DB240.DBX  185.3;
      =     DB240.DBX  265.3;
      =     DB240.DBX  345.3;
      =     DB240.DBX  425.3;
      =     DB240.DBX  505.3;
      =     DB240.DBX  585.3;
      =     DB240.DBX  665.3;
      =     DB240.DBX  745.3;
      =     DB240.DBX  825.3;
NETWORK
TITLE =Special Input

      A     #U.Seq.Sim;
      =     DB241.DBX   81.3;

NETWORK
TITLE =Counter

      A     #U.Seq.Sim;
      A     M    101.0;


      CLR   ;
NETWORK
TITLE =Analog Input

      A     #U.Seq.Sim;

NETWORK
TITLE =Universal Value

      A     #U.Seq.Sim;
//      =     "C04UnVD".unv001.Sim;
//      =     "C04UnVD".unv002.Sim;
//      =     "C04UnVD".unv003.Sim;
//      =     "C04UnVD".unv004.Sim;

NETWORK
TITLE =PID

      A     #U.Seq.Sim;

NETWORK
TITLE =Message

      A     #U.Seq.Sim;
//      =     "C04MsgD".msg001.Sim;
//      =     "C04MsgD".msg002.Sim;
//      =     "C04MsgD".msg003.Sim;

NETWORK
TITLE =VLT

      A     #U.Seq.Sim;

END_FUNCTION_BLOCK

FUNCTION_BLOCK FB 151
TITLE =C05: Syrup Transfer x
// NW  1 : phase and index evaluation
// NW  2 : phase  1: start position
// NW  3 : phase  3: Prerinse
// NW  4 : phase  4: Fill System
// NW  5 : phase  5: Transfer
// NW  6 : phase  8: Push Out
// NW  7 : phase 11: Postrinse
// NW  8 : phase 18: Send Mole
// NW  9 : phase 19: Return Mole
// NW 10 : phase 21: Prepare Line
// NW 11 : phase 22: Tank Selection
// NW 12 : phase 30: CIP Active
// NW 13 : phase 31: CIP Start
// NW 14 : phase 32: CIP Push Out
// NW 15 : phase 34: CIP Rinsing
// NW 16 : phase 36: CIP Drain
// NW 17 : phase 40: CIP End
// NW 18 : end of sequence
// NW 19 : unit hold request
//SFM   Use                                 Datatype        UoM
//----+-------------------------------------------------------------------------
// 09 : Process Time                        Duration        min
// 40 : Density                             Value           kg/l
// 42 : Material                            Value
// 43 : Source                              Value
// 44 : Standby                             Value
AUTHOR : Woermann
NAME : C05Seq
VERSION : 0.1
CODE_VERSION1


VAR
  U : UDT 151;
END_VAR
VAR_TEMP
  CIP : BOOL ;	//CIP active
  ComCIP : BOOL ;	//Communication With CIP Active
  RRel : BOOL ;	//Run Release
  EStopOK : BOOL ;	//emergency OK
  StepMax : BOOL ;	//StepMax (last) active
  SubStepMax : BOOL ;	//SubStepMax (last) active
  SubStepMaxD : BOOL ;	//SubStepMax (last) done
  ChkOK : BOOL ;	//SubStepMax (last) done
  xTmp : BOOL ;	//Temporary BOOL (free for general use)
  iTmp : INT ;	//Temporary INT (free for general use)
  dTmp : DINT ;	//Temporary DINT (free for general use)
  rTmp : REAL ;	//Temporary REAL (free for general use)
  dUnitNo : DINT ;	//Unit Number
  UnitNo : INT ;	//Unit Number
  EquipmentID : INT ;	//Equipment ID
  S2I : STRUCT 	//SFM to indexes
   SFM26 : STRUCT 	//Cip Step On Condition
    I00 : BOOL ;	//Please Select
    I01 : BOOL ;	//Conductivity High
    I02 : BOOL ;	//Conductivity Low
    I03 : BOOL ;	//Time
    I04 : BOOL ;	//Amount
    I05 : BOOL ;	//Temperature High
    I06 : BOOL ;	//Temperature Low
    I07 : BOOL ;
    I08 : BOOL ;
    I09 : BOOL ;
    I10 : BOOL ;
    I11 : BOOL ;
    I12 : BOOL ;
    I13 : BOOL ;
    I14 : BOOL ;
    I15 : BOOL ;
    I16 : BOOL ;
    I17 : BOOL ;
    I18 : BOOL ;
    I19 : BOOL ;
    I20 : BOOL ;
    I21 : BOOL ;
    I22 : BOOL ;
    I23 : BOOL ;
    I24 : BOOL ;
    I25 : BOOL ;
    I26 : BOOL ;
    I27 : BOOL ;
    I28 : BOOL ;
    I29 : BOOL ;
    I30 : BOOL ;
    I31 : BOOL ;
   END_STRUCT ;
   SFM27 : STRUCT 	//Cip Prerun
    I00 : BOOL ;	//None
    I01 : BOOL ;	//Recovered Water
    I02 : BOOL ;	//Caustic
    I03 : BOOL ;
    I04 : BOOL ;	//Acid
    I05 : BOOL ;
    I06 : BOOL ;
    I07 : BOOL ;
    I08 : BOOL ;
    I09 : BOOL ;
    I10 : BOOL ;
    I11 : BOOL ;
    I12 : BOOL ;	//Fresh Water
    I13 : BOOL ;	//Warm Water
    I14 : BOOL ;
    I15 : BOOL ;
    I16 : BOOL ;
    I17 : BOOL ;
    I18 : BOOL ;
    I19 : BOOL ;
    I20 : BOOL ;
    I21 : BOOL ;
    I22 : BOOL ;
    I23 : BOOL ;
    I24 : BOOL ;
    I25 : BOOL ;
    I26 : BOOL ;
    I27 : BOOL ;
    I28 : BOOL ;
    I29 : BOOL ;
    I30 : BOOL ;
    I31 : BOOL ;
   END_STRUCT ;
   SFM28 : STRUCT 	//Cip Return
    I00 : BOOL ;	//None
    I01 : BOOL ;	//Recovered Water
    I02 : BOOL ;	//Caustic
    I03 : BOOL ;
    I04 : BOOL ;	//Acid
    I05 : BOOL ;
    I06 : BOOL ;
    I07 : BOOL ;
    I08 : BOOL ;
    I09 : BOOL ;
    I10 : BOOL ;
    I11 : BOOL ;
    I12 : BOOL ;	//Fresh Water
    I13 : BOOL ;	//Warm Water
    I14 : BOOL ;
    I15 : BOOL ;	//Drain
    I16 : BOOL ;
    I17 : BOOL ;
    I18 : BOOL ;
    I19 : BOOL ;
    I20 : BOOL ;
    I21 : BOOL ;
    I22 : BOOL ;
    I23 : BOOL ;
    I24 : BOOL ;
    I25 : BOOL ;
    I26 : BOOL ;
    I27 : BOOL ;
    I28 : BOOL ;
    I29 : BOOL ;
    I30 : BOOL ;
    I31 : BOOL ;
   END_STRUCT ;
   SFM37 : STRUCT 	//Cip Pump Mode
    I00 : BOOL ;	//Off
    I01 : BOOL ;	//Flow
    I02 : BOOL ;	//Pressure
    I03 : BOOL ;	//Fix Speed
    I04 : BOOL ;
    I05 : BOOL ;
    I06 : BOOL ;
    I07 : BOOL ;
    I08 : BOOL ;
    I09 : BOOL ;
    I10 : BOOL ;
    I11 : BOOL ;
    I12 : BOOL ;
    I13 : BOOL ;
    I14 : BOOL ;
    I15 : BOOL ;
    I16 : BOOL ;
    I17 : BOOL ;
    I18 : BOOL ;
    I19 : BOOL ;
    I20 : BOOL ;
    I21 : BOOL ;
    I22 : BOOL ;
    I23 : BOOL ;
    I24 : BOOL ;
    I25 : BOOL ;
    I26 : BOOL ;
    I27 : BOOL ;
    I28 : BOOL ;
    I29 : BOOL ;
    I30 : BOOL ;
    I31 : BOOL ;
   END_STRUCT ;
   SFM31 : STRUCT 	//Cip Distribution Circuit No
    I00 : BOOL ;	//Please Select
    I01 : BOOL ;	//Auto Select
    I02 : BOOL ;
    I03 : BOOL ;
    I04 : BOOL ;
    I05 : BOOL ;
    I06 : BOOL ;
    I07 : BOOL ;
    I08 : BOOL ;
    I09 : BOOL ;
    I10 : BOOL ;
    I11 : BOOL ;
    I12 : BOOL ;
    I13 : BOOL ;
    I14 : BOOL ;
    I15 : BOOL ;
    I16 : BOOL ;
    I17 : BOOL ;
    I18 : BOOL ;
    I19 : BOOL ;
    I20 : BOOL ;
    I21 : BOOL ;
    I22 : BOOL ;
    I23 : BOOL ;
    I24 : BOOL ;
    I25 : BOOL ;
    I26 : BOOL ;
    I27 : BOOL ;
    I28 : BOOL ;
    I29 : BOOL ;
    I30 : BOOL ;
    I31 : BOOL ;
   END_STRUCT ;
   SFM13 : STRUCT 	//Cip Step On Condition
    I00 : BOOL ;	//Auto
    I01 : BOOL ;	//Schalter
    I02 : BOOL ;	//Auto und Schalter
    I03 : BOOL ;	//Auto oder Schalter
    I04 : BOOL ;
    I05 : BOOL ;
    I06 : BOOL ;
    I07 : BOOL ;
    I08 : BOOL ;
    I09 : BOOL ;
    I10 : BOOL ;
    I11 : BOOL ;
    I12 : BOOL ;
    I13 : BOOL ;
    I14 : BOOL ;
    I15 : BOOL ;
    I16 : BOOL ;
    I17 : BOOL ;
    I18 : BOOL ;
    I19 : BOOL ;
    I20 : BOOL ;
    I21 : BOOL ;
    I22 : BOOL ;
    I23 : BOOL ;
    I24 : BOOL ;
    I25 : BOOL ;
    I26 : BOOL ;
    I27 : BOOL ;
    I28 : BOOL ;
    I29 : BOOL ;
    I30 : BOOL ;
    I31 : BOOL ;
   END_STRUCT ;
  END_STRUCT ;
  ComXYZ : BOOL ;
  ComSRC : BOOL ;	//Communication with SRC Syrup
  ComDST : BOOL ;	//Communication with DST
  ComWater : BOOL ;	//Communication with Water Transfer to Syrup
END_VAR
BEGIN
NETWORK
TITLE = Phase and Index Evaluation

      CLR   ;
      =     #RRel;
      =     DB155.DBX   27.2;

// ---------------------------------------------------------------------------
// write max used SFM's (last SFM number + 1)
      L     60;
      T     #U.SFMQuant;

// ---------------------------------------------------------------------------
// unit & equipment number
      L     MB   112;
      T     #UnitNo;

      L     DB155.DBW   14;
      L     1000;
      *I    ;
      L     #UnitNo;
      +I    ;
      T     #EquipmentID;

// ---------------------------------------------------------------------------
// CIP active
      L     MW   114;
      L     0;
      <I    ;
      =     #CIP;

// ---------------------------------------------------------------------------
// communicating units
      L     MD   124;
      L     DB155.DBD  346;
      ==D   ;
//      A     #CIP
      =     #ComCIP;

      L     MD   124;
//      L     "UxxxComD".Own.PrId //!!! Fill in Communicating Unit Number
      ==D   ;
      =     #ComXYZ; //!!! Fill in Shortname for Communicating Unit

// Source
      L     MD   124;
      L     DB155.DBD  250;
      ==D   ;
      CLR   ;
      A(    ;
      L     #U.Seq.SFM[42].Sp; // Material
      L     DB155.DBD  270;
      ==R   ;
      )     ;
      SET   ;
      =     #ComSRC;

// Destination
      AN    DB155.DBX  312.7;
      SET   ;
      =     #ComDST;

// Water Transfer Syrup
      A     DB1595.DBX   26.3; // Run Release
      =     #ComWater;

      O     M    120.7;
      O     #CIP;
      O     #ComWater;
      JC    M902;
      L     902; // Wasserversorgung überprüfen!
      T     MD    90;
M902: NOP   0;

// ---------------------------------------------------------------------------
// process timer start
      SET   ;
      =     M    131.0;

// ---------------------------------------------------------------------------
// emergency OK
      A     DB155.DBX   27.0;
      =     #EStopOK;

// define last (Sub)Step active
      L     #U.Seq.StepMax;
      L     MW   104;
      ==I   ;
      =     #StepMax;

      L     #U.Seq.SubStepMax;
      L     MW   118;
      ==I   ;
      =     #SubStepMax;

      A     #SubStepMax;
      A     #U.Seq.SPD;
      AN    M    103.2;
      =     #SubStepMaxD;

// ---------------------------------------------------------------------------
// phase evaluation
      L     MW   108;
      JL    X0;
      JU    X0; // phase  0:
      JU    X1; // phase  1: start position
      JU    X0; // phase  2:
      JU    X3; // phase  3: Prerinse
      JU    X4; // phase  4: Fill System
      JU    X5; // phase  5: Transfer
      JU    X0; // phase  6:
      JU    X0; // phase  7:
      JU    X8; // phase  8: Push Out
      JU    X0; // phase  9:
      JU    X0; // phase 10:
      JU    X11; // phase 11: Postrinse
      JU    X0; // phase 12:
      JU    X13; // phase 13: Ende
      JU    X0; // phase 14:
      JU    X0; // phase 15:
      JU    X0; // phase 16:
      JU    X0; // phase 17:
      JU    X18; // phase 18: Send Mole
      JU    X19; // phase 19: Return Mole
      JU    X0; // phase 20:
      JU    X21; // phase 21: Prepare Line
      JU    X22; // phase 22: Tank Selection
      JU    X0; // phase 23:
      JU    X0; // phase 24:
      JU    X0; // phase 25:
      JU    X0; // phase 26:
      JU    X0; // phase 27:
      JU    X0; // phase 28:
      JU    X0; // phase 29:
      JU    X30; // phase 30: CIP Passive
      JU    X31; // phase 31: CIP Start
      JU    X32; // phase 32: CIP Push Out
      JU    X0; // phase 33:
      JU    X34; // phase 34: CIP Rinsing
      JU    X0; // phase 35:
      JU    X36; // phase 36: CIP Drain
      JU    X0; // phase 37:
      JU    X0; // phase 38:
      JU    X0; // phase 39:
      JU    X40; // phase 40: CIP End
X0:   SET   ;
      S     M    108.7; // Error unknown phase
      JU    COMM;
NETWORK
TITLE =phase 1: startposition

X1:   SET   ;

// ---------------------------------------------------------------------------
// general functions
// ---------------------------------------------------------------------------
// reset signals
      A     M    102.2;
      R     #U.Seq.Switch.Sw1;
      R     #U.Seq.Switch.Sw2;
      R     #U.Seq.User.Bit12;
      R     #U.Seq.User.Bit13;

      AN    M    102.0;
      =     M    161.0; // Reset Process Timer

      CALL FC   709 (// Reset "Simulation" And "Ignore"
           UnitNo                   := #UnitNo,// Of All Control Modules
           Enable                   := M    102.2);// At First Cycle of Startposition (Idle)

// MolchSignale für Sirupraum
      A     DB251.DBX  378.7;
      O     DB251.DBX  438.7;
      =     DB250.DBX 3708.2;

      A     DB251.DBX  978.7;
      O     DB251.DBX 1038.7;
      =     DB250.DBX 3788.2;
      =     DB250.DBX 1708.2;

      A     DB250.DBX 3788.2;
      A     M    102.3;
      =     DB250.DBX 3948.0;

// ---------------------------------------------------------------------------
// start check --------------------------------------------------------------
      A     #CIP;
      JC    M010;

      CALL FC   150 (
           ChkType                  := 1,// production
           ChkOK                    := M    122.0);
      JU    COMM;

M010: CALL FC   150 (
           ChkType                  := 2,// CIP
           ChkOK                    := M    122.0);
      JU    COMM;
NETWORK
TITLE =phase 3: Prerinse
//SFM   Use                                 Datatype        UoM
//----+-------------------------------------------------------------------------
// 00 : Watch Dog Time                      Duration        min
// 20 : Flow                                Value           l/h
// 41 : Amount                              Value           kg
X3:   SET   ;
// ---------------------------------------------------------------------------
// General CM evaluation
      CALL FC   150 (
           ChkType                  := 3,
           ChkOK                    := #ChkOK);

      AN    #ChkOK;
      S     M    120.3;

// ---------------------------------------------------------------------------
// general functions
      AN    M    121.2;
      A     M    102.3;
      =     #RRel;

// ---------------------------------------------------------------------------
// messages
// ---------------------------------------------------------------------------
// timer & counter
      A     M    102.0;

// ---------------------------------------------------------------------------
// pause timer
// ---------------------------------------------------------------------------
// communication

// ---------------------------------------------------------------------------
// control modules
      A     M    102.3;

// ---------------------------------------------------------------------------
// transition condition
      A     #SubStepMaxD;
      =     M    102.1;

// subphase evaluation
      L     MW   110;
      JL    A300;
      JU    COMM; // subphase  0:
// ---------------------------------------------------------------------------
A300: SET   ;
      S     M    110.7; // Error unknown subphase
      JU    COMM;
NETWORK
TITLE =phase 4: Fill System
//SFM   Use                                 Datatype        UoM
//----+-------------------------------------------------------------------------
// 00 : Watch Dog Time                      Duration        min
// 20 : Flow                                Value           l/h
// 41 : Amount                              Value           kg
X4:   SET   ;
// ---------------------------------------------------------------------------
// General CM evaluation
      CALL FC   150 (
           ChkType                  := 3,
           ChkOK                    := #ChkOK);

      AN    #ChkOK;
      S     M    120.3;

// ---------------------------------------------------------------------------
// general functions
      AN    M    121.2;
      A     M    102.3;
      =     #RRel;

// ---------------------------------------------------------------------------
// messages
// ---------------------------------------------------------------------------
// timer & counter
      A     M    102.0;

// ---------------------------------------------------------------------------
// pause timer
// ---------------------------------------------------------------------------
// communication

// ---------------------------------------------------------------------------
// control modules
      A     M    102.3;

// ---------------------------------------------------------------------------
// transition condition
      SET   ;
      AN    M    102.2; // Batch buffer full when mole in returned position
      =     M    102.1;

// subphase evaluation
      L     MW   110;
      JL    A400;
      JU    COMM; // subphase  0:
// ---------------------------------------------------------------------------
A400: SET   ;
      S     M    110.7; // Error unknown subphase
      JU    COMM;
NETWORK
TITLE =phase 5: Transfer
//SFM   Use                                 Datatype        UoM
//----+-------------------------------------------------------------------------
// 00 : Watch Dog Time                      Duration        min
// 20 : Flow                                Value           l/h
// 41 : Amount                              Value           kg
X5:   SET   ;
// ---------------------------------------------------------------------------
// General CM evaluation
      CALL FC   150 (
           ChkType                  := 3,
           ChkOK                    := #ChkOK);

      AN    #ChkOK;
      S     M    120.3;

// ---------------------------------------------------------------------------
// index evaluation: CIP Step On Condition
      CALL FC    45 (
           SFM                      := #U.Seq.SFM[13].Sp,
           Indexes                  := #S2I.SFM13);

// ---------------------------------------------------------------------------
// general functions
      AN    M    121.2;
      A     M    102.3;
      =     #RRel;

// ---------------------------------------------------------------------------
// messages
// ---------------------------------------------------------------------------
// timer & counter
      A     M    102.0;

// ---------------------------------------------------------------------------
// pause timer
// ---------------------------------------------------------------------------
// communication
// MolchSignale für Sirupraum
      A     DB251.DBX  378.7;
      O     DB251.DBX  438.7;
      =     DB250.DBX 3708.2;

      A     DB251.DBX  978.7;
      O     DB251.DBX 1038.7;
      =     DB250.DBX 3788.2;

      A     M    102.3;
      =     DB250.DBX 3868.0;

// ---------------------------------------------------------------------------
// control modules
      A     M    102.3;
      CLR   ;

// ---------------------------------------------------------------------------
// transition condition
      L     DB155.DBD  250;
      L     MD   124;

      O(    ;
      A     DB155.DBX  269.0;
      A     #S2I.SFM13.I00;
      )     ;
      O(    ;
      A     #U.Seq.Switch.Sw1; // Start SR -> A7
      A     #S2I.SFM13.I01;
      )     ;
      O(    ;
      A     #U.Seq.Switch.Sw1; // Start SR -> A7
      A     DB155.DBX  269.0;
      A     #S2I.SFM13.I02;
      )     ;
      O(    ;
      A     #U.Seq.Switch.Sw1; // Start SR -> A7
      O     DB155.DBX  269.0;
      A     #S2I.SFM13.I03;
      )     ;
      =     M    102.1;

// ---------------------------------------------------------------------------
// ---------------------------------------------------------------------------
// subphase repeat function
      A     #SubStepMax;
      JCN   Y5;
      L     1;
      T     MW   116;
Y5:   SET   ;

// subphase evaluation
      L     MW   110;
      JL    A500;
      JU    COMM; // subphase  0:
      JU    A501; // subphase  1: Waiting
      JU    A502; // subphase  2: Active
      JU    A503; // subphase  3: Tank Change
// ---------------------------------------------------------------------------
A500: SET   ;
      S     M    110.7; // Error unknown subphase
      JU    COMM;

// subphase 1: Waiting
A501: SET   ;
      A     M    103.3;
      =     DB155.DBX   26.3;
      =     DB155.DBX   26.0;
// -------------------------------------------------
// subphase timer & counter
      A     M    103.0;

// -------------------------------------------------
// subphase actuator
      A     M    103.3;

// -------------------------------------------------
// subphase transition
      A     DB155.DBX  314.1;
//   A     "C05ComD".SRC.WfEm
      =     M    103.1;
      JU    COMM;

// subphase 2: Active
A502: SET   ;
      A     M    103.3;
      =     DB155.DBX   26.4;
      =     DB155.DBX   26.1;
// -------------------------------------------------
// subphase timer & counter
      A     M    103.0;

// -------------------------------------------------
// subphase actuator
      A     M    103.3;

// -------------------------------------------------
// subphase transition
//  AN    "C05ComD".SRC.Emti
// ON    "C05ComD".SRC.WfEm
      AN    DB155.DBX  314.1;
      AN    M    103.2;
      =     M    103.1;
      JU    COMM;

// subphase 3: Tank Change
A503: SET   ;

// -------------------------------------------------
// subphase timer & counter
      A     M    103.0;

// -------------------------------------------------
// subphase actuator
      A     M    103.3;

// -------------------------------------------------
// subphase transition
      CLR   ;
      =     M    103.1;
      JU    COMM;
NETWORK
TITLE =phase 8: Push Out
//SFM   Use                                 Datatype        UoM
//----+-------------------------------------------------------------------------
// 00 : Watch Dog Time                      Duration        min
// 20 : Flow                                Value           l/h
// 41 : Amount                              Value           kg
X8:   SET   ;
// ---------------------------------------------------------------------------
// General CM evaluation
      CALL FC   150 (
           ChkType                  := 3,
           ChkOK                    := #ChkOK);

      AN    #ChkOK;
      S     M    120.3;

// ---------------------------------------------------------------------------
// general functions
      AN    M    121.2;
      A     M    102.3;
      =     #RRel;

// ---------------------------------------------------------------------------
// messages
// ---------------------------------------------------------------------------
// timer & counter
      A     M    102.0;

// ---------------------------------------------------------------------------
// pause timer
// ---------------------------------------------------------------------------
// communication

// ---------------------------------------------------------------------------
// control modules
      A     M    102.3;

// ---------------------------------------------------------------------------
// transition condition
      SET   ;
      =     M    102.1;

// subphase evaluation
      L     MW   110;
      JL    A800;
      JU    COMM; // subphase  0:
// ---------------------------------------------------------------------------
A800: SET   ;
      S     M    110.7; // Error unknown subphase
      JU    COMM;
NETWORK
TITLE =phase 11: Postrinse
//SFM   Use                                 Datatype        UoM
//----+-------------------------------------------------------------------------
// 00 : Watch Dog Time                      Duration        min
// 20 : Flow                                Value           l/h
// 41 : Amount                              Value           kg
X11:  SET   ;
// ---------------------------------------------------------------------------
// General CM evaluation
      CALL FC   150 (
           ChkType                  := 3,
           ChkOK                    := #ChkOK);

      AN    #ChkOK;
      S     M    120.3;

// ---------------------------------------------------------------------------
// general functions
      AN    M    121.2;
      A     M    102.3;
      =     #RRel;

// ---------------------------------------------------------------------------
// messages
// ---------------------------------------------------------------------------
// timer & counter
      A     M    102.0;

// ---------------------------------------------------------------------------
// pause timer
// ---------------------------------------------------------------------------
// communication
// MolchSignale für Sirupraum
      A     DB251.DBX  978.7;
      O     DB251.DBX 1038.7;
      =     DB250.DBX 3788.2;
      =     DB250.DBX 1708.2;

// ---------------------------------------------------------------------------
// control modules
      A     M    102.3;

// ---------------------------------------------------------------------------
// transition condition
      A     #SubStepMaxD;
      =     M    102.1;

// subphase evaluation
      L     MW   110;
      JL    B100;
      JU    COMM; // subphase  0:
// ---------------------------------------------------------------------------
B100: SET   ;
      S     M    110.7; // Error unknown subphase
      JU    COMM;
NETWORK
TITLE =phase 13: Ende
//SFM   Use                                 Datatype        UoM
//----+-------------------------------------------------------------------------
// 00 : Watch Dog Time                      Duration        min
// 20 : Flow                                Value           l/h
// 41 : Amount                              Value           kg
X13:  SET   ;
// ---------------------------------------------------------------------------
// General CM evaluation
      CALL FC   150 (
           ChkType                  := 3,
           ChkOK                    := #ChkOK);

      AN    #ChkOK;
      S     M    120.3;

// ---------------------------------------------------------------------------
// general functions
      AN    M    121.2;
      A     M    102.3;
      =     #RRel;

// ---------------------------------------------------------------------------
// messages
// ---------------------------------------------------------------------------
// timer & counter

// ---------------------------------------------------------------------------
// pause timer
// ---------------------------------------------------------------------------
// communication
// MolchSignale für Sirupraum
// Endposition
      A     DB251.DBX  978.7;
      O     DB251.DBX 1038.7;
      A     M    103.3;
      =     DB250.DBX 1708.0;

// ---------------------------------------------------------------------------
// control modules
      A     M    102.3;

// ---------------------------------------------------------------------------
// transition condition
      L     DB155.DBD  346;
      L     MD   124;
      <>D   ;
      O     DB155.DBX  360.7;
      AN    M    102.2;
      =     M    102.1;

// subphase evaluation
      L     MW   110;
      JL    B300;
      JU    COMM; // subphase  0:
// ---------------------------------------------------------------------------
B300: SET   ;
      S     M    110.7; // Error unknown subphase
      JU    COMM;
NETWORK
TITLE =phase 18: Send Mole
//SFM   Use                                 Datatype        UoM
//----+-------------------------------------------------------------------------
// 00 : Watch Dog Time                      Duration        min
// 05 : Step Time                           Duration        s
// 06 : Delay Time                          Duration        s
X18:  SET   ;
// ---------------------------------------------------------------------------
// General CM evaluation
      CALL FC   150 (
           ChkType                  := 3,
           ChkOK                    := #ChkOK);

      AN    #ChkOK;
      S     M    120.3;

      AN    M    102.0;
      R     #U.Seq.Switch.Sw1;

// ---------------------------------------------------------------------------
// general functions
      AN    M    121.2;
      A     M    102.3;
      =     #RRel;

      AN    M    102.0;
      R     #U.Seq.Switch.Sw1;
// ---------------------------------------------------------------------------
// messages
// ---------------------------------------------------------------------------
// timer & counter
      A     M    102.0;

// ---------------------------------------------------------------------------
// pause timer
      AN    M    102.3;
      O     M    150.4;
      S     M    140.4; // Step Time

      AN    M    102.3;
      O     M    150.5;
      S     M    140.5; // Delay Time

// ---------------------------------------------------------------------------
// communication
      A     M    102.3;
      S     DB155.DBX   27.2;

      A     M    102.0;
      =     DB250.DBX 1628.0;

// MolchSignale für Sirupraum
      A     DB251.DBX  378.7;
      O     DB251.DBX  438.7;
      =     DB250.DBX 3708.2;

      A     DB251.DBX  978.7;
      O     DB251.DBX 1038.7;
      =     DB250.DBX 3788.2;

// ---------------------------------------------------------------------------
// control modules
      A     M    102.3;

// ---------------------------------------------------------------------------
// transition condition
      A     #SubStepMaxD;
      =     M    102.1;

// ---------------------------------------------------------------------------
// ---------------------------------------------------------------------------
// subphase repeat function
//      A     #SubStepMax
//      JCN  Y18
//      L     1
//      T     "SOSubStepNew"
//Y18:  SET

// subphase evaluation
      L     MW   110;
      JL    B800;
      JU    COMM; // subphase  0:
      JU    B801; // subphase  1: Open Horns
      JU    B802; // subphase  2: Raise Baskets
      JU    B803; // subphase  3: Send Mole
      JU    B804; // subphase  4: Lower Baskets
      JU    B805; // subphase  5: Line Rinsing
      JU    B806; // subphase  6: Depressurise
      JU    B807; // subphase  7: End
// ---------------------------------------------------------------------------
B800: SET   ;
      S     M    110.7; // Error unknown subphase
      JU    COMM;

// subphase 1: Open Horns
B801: SET   ;

// -------------------------------------------------
// subphase timer & counter
      A     DB250.DBX  502.6;
      A     DB250.DBX  582.6;
      A     DB250.DBX  582.6;
      A     DB250.DBX 1382.6;
      A     M    103.0;
      =     M    130.5; // Delay Time
// -------------------------------------------------
// subphase actuator
// Horns
      A     M    103.0;
      =     DB250.DBX  508.0;
      =     DB250.DBX  588.0;
      =     DB250.DBX 1308.0;
      =     DB250.DBX 1388.0;

// -------------------------------------------------
// subphase transition
      A     M    150.5; // Delay TIme
      AN    M    103.2;
      =     M    103.1;
      JU    COMM;

// subphase 2: Raise Baskets
B802: SET   ;

// -------------------------------------------------
// subphase timer & counter
      A     DB251.DBX  258.7;
      A     DB251.DBX  858.7;
      CLR   ; // Signale gehen nicht
      A     DB250.DBX  342.6;
      A     DB250.DBX 1142.6;
      A     M    103.0;
      =     M    130.5; // Delay Time
// -------------------------------------------------
// subphase actuator
// Horns
      A     M    103.0;
      =     DB250.DBX  508.0;
      =     DB250.DBX  588.0;
      =     DB250.DBX 1308.0;
      =     DB250.DBX 1388.0;

// Basktets
      A     M    102.3;
      =     DB250.DBX  348.0;
      =     DB250.DBX 1148.0;

// -------------------------------------------------
// subphase transition
      A     M    150.5; // Delay Time
      =     M    103.1;
      JU    COMM;

// subphase 3: Send Mole
B803: SET   ;

// -------------------------------------------------
// subphase timer & counter
      A     DB251.DBX  978.7;
      O     DB251.DBX 1038.7;
      A     M    103.0;
      =     M    130.5; // Delay Time
// -------------------------------------------------
// subphase actuator
// Horns
      A     M    103.0;
      =     DB250.DBX  508.0;
      =     DB250.DBX  588.0;
      =     DB250.DBX 1308.0;
      =     DB250.DBX 1388.0;

// Basktets
      A     M    102.3;
      =     DB250.DBX  348.0;
      =     DB250.DBX 1148.0;

// Water
      A     M    103.3;
      =     DB250.DBX  188.0;

// -------------------------------------------------
// subphase transition
      A     M    150.5; // Delay time
      =     M    103.1;
      JU    COMM;

// subphase 4: Lower Baskets
B804: SET   ;

// -------------------------------------------------
// subphase timer & counter
      A     DB251.DBX  318.7;
      A     DB251.DBX  918.7;
      CLR   ;
      A     DB250.DBX  422.6;
      A     DB250.DBX 1222.6;
      A     M    103.0;
      =     M    130.5; // Delay Time
// -------------------------------------------------
// subphase actuator
// Horns
      A     M    103.0;
      =     DB250.DBX  508.0;
      =     DB250.DBX  588.0;
      =     DB250.DBX 1308.0;
      =     DB250.DBX 1388.0;

// Basktets
      A     M    102.3;
      =     DB250.DBX  428.0;
      =     DB250.DBX 1228.0;

// Drain
      A     M    103.3;
      =     DB250.DBX 1068.0;

// Endposition
      A     M    103.3;
      =     DB250.DBX 1708.0;

// Water
      A     M    103.3;
      =     DB250.DBX  188.0;

// -------------------------------------------------
// subphase transition
      A     M    150.5; // Delay Time
      =     M    103.1;
      JU    COMM;

// subphase 5: Line Rinsing
B805: SET   ;

// -------------------------------------------------
// subphase timer & counter
      A     M    103.0;
      =     M    130.4; // Step Time
// -------------------------------------------------
// subphase actuator

// Drain
      A     M    103.3;
      =     DB250.DBX 1068.0;

// Endposition
      A     M    103.3;
      =     DB250.DBX 1708.0;

// Water
      A     M    103.3;
      =     DB250.DBX  188.0;

// -------------------------------------------------
// subphase transition
      A     M    150.4; // Step Time
      =     M    103.1;
      JU    COMM;

// subphase 6: Depressurise
B806: SET   ;

// -------------------------------------------------
// subphase timer & counter
      A     M    103.0;
      =     M    130.4; // Step Time
// -------------------------------------------------
// subphase actuator

// Drain
      A     M    103.3;
      =     DB250.DBX 1068.0;

// Endposition
      A     M    103.3;
      =     DB250.DBX 1708.0;

// -------------------------------------------------
// subphase transition
      A     M    150.4; // Step Time
      =     M    103.1;
      JU    COMM;

// subphase 7: End
B807: SET   ;

// -------------------------------------------------
// subphase timer & counter
      A     M    103.0;
      =     M    130.4; // Step Time
// -------------------------------------------------
// subphase actuator
      A     M    103.3;

// -------------------------------------------------
// subphase transition
      A     M    150.4; // Step Time
      =     M    103.1;
      JU    COMM;
NETWORK
TITLE =phase 19: Return Mole
//SFM   Use                                 Datatype        UoM
//----+-------------------------------------------------------------------------
// 00 : Watch Dog Time                      Duration        min
// 05 : Step Time                           Duration        s
// 06 : Delay Time                          Duration        s
X19:  SET   ;
// ---------------------------------------------------------------------------
// General CM evaluation
      CALL FC   150 (
           ChkType                  := 3,
           ChkOK                    := #ChkOK);

      AN    #ChkOK;
      S     M    120.3;

      L     MB   112;
      L     103; // No automict return with KEG
      <>I   ;
      A     M    102.2;
      S     #U.Seq.Switch.Sw2;

      AN    M    102.0;
      R     #U.Seq.Switch.Sw2;


// ---------------------------------------------------------------------------
// general functions
      AN    M    121.2;
      A     M    102.3;
      =     #RRel;

      AN    M    102.0;
      R     #U.Seq.User.Bit12;
      R     #U.Seq.User.Bit13;

// ---------------------------------------------------------------------------
// messages
// ---------------------------------------------------------------------------
// timer & counter
      A     M    102.0;

// ---------------------------------------------------------------------------
// pause timer
      AN    M    102.3;
      O     M    150.4;
      S     M    140.4; // Step Time

      AN    M    102.3;
      O     M    150.5;
      S     M    140.5; // Delay Time

// ---------------------------------------------------------------------------
// communication
// MolchSignale für Sirupraum
      A     DB251.DBX  378.7;
      O     DB251.DBX  438.7;
      =     DB250.DBX 3708.2;

      A     DB251.DBX  978.7;
      O     DB251.DBX 1038.7;
      =     DB250.DBX 3788.2;


// ---------------------------------------------------------------------------
// control modules
      A     M    102.3;

// ---------------------------------------------------------------------------
// transition condition
      A     #U.Seq.SPO.B1; // Subphase 1
      A     DB251.DBX  378.7;
      A     DB251.DBX  438.7;
      =     #xTmp;

      A     #xTmp;
      O     #SubStepMaxD;
      AN    M    102.2;
      =     M    102.1;

// ---------------------------------------------------------------------------
// ---------------------------------------------------------------------------
// subphase repeat function
//      A     #SubStepMax
//      JCN  Y19
//      L     1
//      T     "SOSubStepNew"
//Y19:  SET

// subphase evaluation
      L     MW   110;
      JL    B900;
      JU    COMM; // subphase  0:
      JU    B901; // subphase  1: Check Mole Position
      JU    B902; // subphase  2: Open Horns
      JU    B903; // subphase  3: Raise Baskets
      JU    B904; // subphase  4: Return Mole
      JU    B905; // subphase  5: Lower Baskets
      JU    B906; // subphase  6: Line Rinsing
      JU    B907; // subphase  7: Depressurise
      JU    B908; // subphase  8: End
// ---------------------------------------------------------------------------
B900: SET   ;
      S     M    110.7; // Error unknown subphase
      JU    COMM;

// subphase 1: Check Mole Position
B901: SET   ;

      AN    DB251.DBX  978.7;
      AN    DB251.DBX 1038.7;
      JCN   N901;
      L     927; // Pig Not Found
      T     MD    90;
N901: NOP   0;
// -------------------------------------------------
// subphase timer & counter


// -------------------------------------------------
// subphase actuator

// -------------------------------------------------
// subphase transition
// Plant
//      A     "C05SpID".GOA_EKEG_3.Sig
//      A     "C05SpID".GOA_EKEG_4.Sig
//      O     "SOStart"
      A     #U.Seq.Switch.Sw2;
      AN    M    103.2;
      =     M    103.1;

      JU    COMM;

// subphase 2: Open Horns
B902: SET   ;

// -------------------------------------------------
// subphase timer & counter

      A     DB250.DBX  502.6;
      A     DB250.DBX  582.6;
      A     DB250.DBX 1302.6;
      A     DB250.DBX 1382.6;
      A     M    103.0;
      =     M    130.5; // Delay Time
// -------------------------------------------------
// subphase actuator
// Horns
      A     M    103.0;
      =     DB250.DBX  508.0;
      =     DB250.DBX  588.0;
      =     DB250.DBX 1308.0;
      =     DB250.DBX 1388.0;

// -------------------------------------------------
// subphase transition
      A     M    150.5; // Delay Time
      AN    M    103.2;
      =     M    103.1;

      JU    COMM;

// subphase 3: Raise Baskets
B903: SET   ;

// -------------------------------------------------
// subphase timer & counter
      A     DB251.DBX  258.7;
      A     DB251.DBX  858.7;
      CLR   ; // Signale gehen nicht
      A     DB250.DBX  342.6;
      A     DB250.DBX 1142.6;
      A     M    103.0;
      =     M    130.5; // Delay Time
// -------------------------------------------------
// subphase actuator
// Horns
      A     M    103.0;
      =     DB250.DBX  508.0;
      =     DB250.DBX  588.0;
      =     DB250.DBX 1308.0;
      =     DB250.DBX 1388.0;


// Basktets
      A     M    102.3;
      =     DB250.DBX  348.0;
      =     DB250.DBX 1148.0;

// -------------------------------------------------
// subphase transition
      A     M    150.5; // Delay Time
      =     M    103.1;
      JU    COMM;

// subphase 4: Return Mole
B904: SET   ;

// -------------------------------------------------
// subphase timer & counter
      A     DB251.DBX  378.7;
      O     DB251.DBX  438.7;
      A     M    103.0;
      =     M    130.5; // Delay Time
// -------------------------------------------------
// subphase actuator
// Horns
      A     M    103.0;
      =     DB250.DBX  508.0;
      =     DB250.DBX  588.0;
      =     DB250.DBX 1308.0;
      =     DB250.DBX 1388.0;


// Basktets
      A     M    102.3;
      =     DB250.DBX  348.0;
      =     DB250.DBX 1148.0;

// Drain
      A     M    103.3;
      =     DB250.DBX  268.0;

// C02
      A     M    103.3;
      =     DB250.DBX  988.0;
      =     DB250.DBX 1068.0;

// -------------------------------------------------
// subphase transition
      A     M    150.5; // Delay Time
      =     M    103.1;
      JU    COMM;

// subphase 5: Lower Baskets
B905: SET   ;
// -------------------------------------------------
// subphase timer & counter
      A     DB251.DBX  318.7;
      A     DB251.DBX  918.7;
      CLR   ;
      A     DB250.DBX  422.6;
      A     DB250.DBX 1222.6;
      A     M    103.0;
      =     M    130.5; // Delay Time
// -------------------------------------------------
// subphase actuator
// Horns
      A     M    103.0;
      =     DB250.DBX  508.0;
      =     DB250.DBX  588.0;
      =     DB250.DBX 1308.0;
      =     DB250.DBX 1388.0;

// Basktets
      A     M    102.3;
      =     DB250.DBX  428.0;
      =     DB250.DBX 1228.0;

// Drain
      A     M    103.3;
      =     DB250.DBX  268.0;

// C02
      A     M    103.3;
      =     DB250.DBX  988.0;
      =     DB250.DBX 1068.0;


// -------------------------------------------------
// subphase transition
      A     M    150.5; // Delay Time
      =     M    103.1;
      JU    COMM;

// subphase 6: Line Rinsing
B906: SET   ;

// -------------------------------------------------
// subphase timer & counter
      A     M    103.0;
      =     M    130.4; // Step Time
// -------------------------------------------------
// Drain
      A     M    103.3;
      =     DB250.DBX  268.0;

// C02
      A     M    103.3;
      =     DB250.DBX  988.0;
      =     DB250.DBX 1068.0;

// -------------------------------------------------
// subphase transition
      A     M    150.4; // Step Time
      =     M    103.1;
      JU    COMM;

// subphase 7: Depressurise
B907: SET   ;

// -------------------------------------------------
// subphase timer & counter
      A     M    103.0;
      =     M    130.4; // Step Time

// -------------------------------------------------
// subphase actuator
// Drain
      A     M    103.3;
      =     DB250.DBX  268.0;

// -------------------------------------------------
// subphase transition
      A     M    150.4; // Step Time
      =     M    103.1;
      JU    COMM;

// subphase 8: End
B908: SET   ;

// -------------------------------------------------
// subphase timer & counter
      A     M    103.0;
      =     M    130.4; // Step Time
// -------------------------------------------------
// subphase actuator
      A     M    103.3;

// -------------------------------------------------
// subphase transition
      A     M    150.4; // Step Time
      =     M    103.1;
      JU    COMM;
NETWORK
TITLE =phase 21: Prepare Line
//SFM   Use                                 Datatype        UoM
//----+-------------------------------------------------------------------------
// 00 : Watch Dog Time                      Duration        min
X21:  SET   ;
// ---------------------------------------------------------------------------
// General CM evaluation
      CALL FC   150 (
           ChkType                  := 3,
           ChkOK                    := #ChkOK);

      AN    #ChkOK;
      S     M    120.3;

// ---------------------------------------------------------------------------
// general functions
      AN    M    121.2;
      A     M    102.3;
      =     #RRel;

// MolchSignale für Sirupraum
      A     DB251.DBX  378.7;
      O     DB251.DBX  438.7;
      =     DB250.DBX 3708.2;

      A     DB251.DBX  978.7;
      O     DB251.DBX 1038.7;
      =     DB250.DBX 3788.2;

// ---------------------------------------------------------------------------
// messages
      AN    #ComSRC;
      JCN   N211;
      L     904; // Source not Ready!
      T     MD    90;
N211: NOP   0;

// ---------------------------------------------------------------------------
// timer & counter
      A     M    102.0;

// ---------------------------------------------------------------------------
// pause timer
// ---------------------------------------------------------------------------
// communication

// ---------------------------------------------------------------------------
// control modules
      A     M    102.3;

// ---------------------------------------------------------------------------
// transition condition
      A     #ComSRC;
      A     #ComDST;
      A     #ComWater;
      =     M    102.1;

// subphase evaluation
      L     MW   110;
      JL    C100;
      JU    COMM; // subphase  0:
// ---------------------------------------------------------------------------
C100: SET   ;
      S     M    110.7; // Error unknown subphase
      JU    COMM;
NETWORK
TITLE =phase 22: Tank Selection
//SFM   Use                                 Datatype        UoM
//----+-------------------------------------------------------------------------
// 00 : Watch Dog Time                      Duration        min
X22:  SET   ;
// ---------------------------------------------------------------------------
// General CM evaluation
      CALL FC   150 (
           ChkType                  := 3,
           ChkOK                    := #ChkOK);

      AN    #ChkOK;
      S     M    120.3;

// ---------------------------------------------------------------------------
// general functions
      AN    M    121.2;
      A     M    102.3;
      =     #RRel;

// ---------------------------------------------------------------------------
// messages
// ---------------------------------------------------------------------------
// timer & counter
      A     M    102.0;

// ---------------------------------------------------------------------------
// pause timer
// ---------------------------------------------------------------------------
// communication

// ---------------------------------------------------------------------------
// control modules
      A     M    102.3;

// ---------------------------------------------------------------------------
// transition condition
      A     #SubStepMaxD;
      =     M    102.1;

// subphase evaluation
      L     MW   110;
      JL    C200;
      JU    COMM; // subphase  0:
// ---------------------------------------------------------------------------
C200: SET   ;
      S     M    110.7; // Error unknown subphase
      JU    COMM;
NETWORK
TITLE =phase 30: CIP Passive
//SFM   Use                                 Datatype        UoM
//----+-------------------------------------------------------------------------
// 00 : Watch Dog Time                      Duration        min
// 05 : Substep Time                        Duration        s
// 22 : Pump Speed                          Value           %
X30:  SET   ;
// ---------------------------------------------------------------------------
// General CM evaluation
      CALL FC   150 (
           ChkType                  := 4,
           ChkOK                    := #ChkOK);

      AN    #ChkOK;
      S     M    120.3;

// ---------------------------------------------------------------------------
// general functions
      AN    M    121.2;
      A     M    102.3;
      =     #RRel;

// ---------------------------------------------------------------------------
// messages
// ---------------------------------------------------------------------------
// timer & counter

// ---------------------------------------------------------------------------
// pause timer
      ON    M    102.3;
      O     M    150.4;
      S     M    140.4; // Substep Time

// ---------------------------------------------------------------------------
// communication
      A     M    102.0;
      =     DB155.DBX   26.0;

      A     DB251.DBX 1338.7;
      O     DB251.DBX 1518.7;
      A     M    102.3;
      =     DB155.DBX   26.1;

// ---------------------------------------------------------------------------
// control modules
      A     #ComCIP;
      A     DB155.DBX  268.3;
      A     M    102.3;
      =     DB250.DBX  188.0;

// ---------------------------------------------------------------------------
// transition condition
      L     DB155.DBD  346;
      L     MD   124;
      <>D   ;
      O     DB155.DBX  360.7;
      AN    #ComCIP;
      =     M    102.1;

// ---------------------------------------------------------------------------
// ---------------------------------------------------------------------------
// subphase repeat function
      A     #SubStepMax;
      JCN   Y30;
      L     1;
      T     MW   116;
Y30:  SET   ;

// subphase evaluation
      L     MW   110;
      JL    D000;
      JU    COMM; // subphase  0:
      JU    D001; // subphase  1: Standby
      JU    D002; // subphase  2: Active
      JU    D003; // subphase  3: Expulse
      JU    D004; // subphase  4: Expulse 2
// ---------------------------------------------------------------------------
D000: SET   ;
      S     M    110.7; // Error unknown subphase
      JU    COMM;

// subphase 1: Standby
D001: SET   ;

// -------------------------------------------------
// subphase timer & counter
      A     M    103.0;

// -------------------------------------------------
// subphase actuator
      A     M    103.3;

// -------------------------------------------------
// subphase transition
      SET   ;
      =     M    103.1;
      JU    COMM;

// subphase 2: Active
D002: SET   ;

// -------------------------------------------------
// subphase timer & counter

// -------------------------------------------------
// subphase actuator

// -------------------------------------------------
// subphase transition
      CLR   ;
      =     M    103.1;
      JU    COMM;

// subphase 3: Expulse
D003: SET   ;

// -------------------------------------------------
// subphase timer & counter
      A     M    103.0;
      =     M    130.4; // Step Time

// -------------------------------------------------
// subphase actuator
      A     DB155.DBX  268.3;
      A     M    103.3;
      =     DB5050.DBX  988.0;
      R     DB5050.DBX 1068.0;

// -------------------------------------------------
// subphase transition
      A     M    150.4; // Step Time Done
      =     M    103.1;
      JU    COMM;

// subphase 4: Expulse 2
D004: SET   ;

// -------------------------------------------------
// subphase timer & counter
      A     M    103.0;
      =     M    130.4; // Step Time

// -------------------------------------------------
// subphase actuator
      A     DB155.DBX  268.3;
      A     M    103.3;
      =     DB5050.DBX  268.0;

// -------------------------------------------------
// subphase transition
      A     M    150.4; // Step Time Done
      =     M    103.1;
      JU    COMM;

NETWORK
TITLE =phase 31: CIP Start
//SFM   Use                                 Datatype        UoM
//----+-------------------------------------------------------------------------
// 00 : Watch Dog Time                      Duration        min
X31:  SET   ;
// ---------------------------------------------------------------------------
// General CM evaluation
      CALL FC   150 (
           ChkType                  := 3,
           ChkOK                    := #ChkOK);

      AN    #ChkOK;
      S     M    120.3;

// ---------------------------------------------------------------------------
// general functions
      AN    M    121.2;
      A     M    102.3;
      =     #RRel;

// ---------------------------------------------------------------------------
// messages
// ---------------------------------------------------------------------------
// timer & counter
      A     M    102.0;

// ---------------------------------------------------------------------------
// pause timer
// ---------------------------------------------------------------------------
// communication

// ---------------------------------------------------------------------------
// control modules
      A     M    102.3;

// ---------------------------------------------------------------------------
// transition condition
      A     #SubStepMaxD;
      =     M    102.1;

// ---------------------------------------------------------------------------
// ---------------------------------------------------------------------------
// subphase repeat function
//      A     #SubStepMax
//      JCN  Y31
//      L     1
//      T     "SOSubStepNew"
//Y31:  SET

// subphase evaluation
      L     MW   110;
      JL    D100;
      JU    COMM; // subphase  0:
      JU    D101; // subphase  1: Wait For CIP
      JU    D102; // subphase  2: Wait For Partner
// ---------------------------------------------------------------------------
D100: SET   ;
      S     M    110.7; // Error unknown subphase
      JU    COMM;

// subphase 1: Wait For CIP
D101: SET   ;

// -------------------------------------------------
// subphase timer & counter
      A     M    103.0;

// -------------------------------------------------
// subphase actuator
      A     M    103.3;

// -------------------------------------------------
// subphase transition
      CLR   ;
      =     M    103.1;
      JU    COMM;

// subphase 2: Wait For Partner
D102: SET   ;

